{attribute 'qualified_only'}
{attribute 'strict'}
TYPE AmpelState :
(
	Init := 0,
	Red,
	Disabled,
	Red_Yellow,
	Green,
	Yellow
);
END_TYPE

(* stored: Version 1.1.0.1, ProductVersion 3.1.4024.13
   DUT AmpelState: Id {2d0a0588-a1ff-4ae4-a992-0eab175996f1} *)
